Universal Robots PolyScope program: base_a.urp

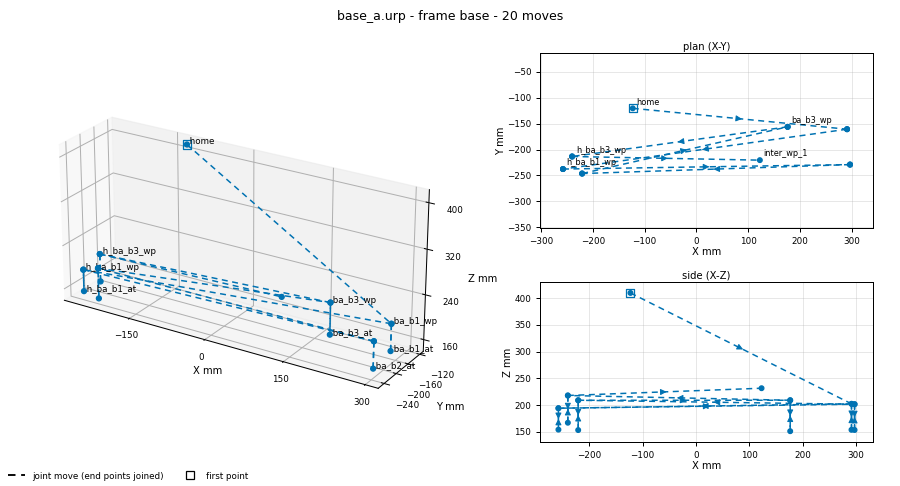
[picture p0: tool path of base_a.urp in frame base, 20 of 20 moves have a stored position in this frame; points joined in program order, loops and branches not executed]
Program base_a (installation=default directory=/programs/Session 1 createdIn=5.3.1.64192 lastSavedIn=5.3.1.64192 robotSerialNumber=20195300365)
Calibrated DH parameters: a=[-0.000093, -0.190649, -0.212673, 0.000091, -0.000205, 0]; d=[0.151591, 44.061648, -42.488068, -1.442789, 0.085322, 0.091911]; alpha=[1.570082, -0.003447, 0.007513, 1.572293, -1.571904, 0]; deltaTheta=[0, -0.672656, 0.728185, -0.055522, 0.000005, 0]
Robot Program (runOnlyOnce=true)
  URCap Gripper Activate (Robotiq_Grippers, Robotiq Inc.) dataModel(ResetAndActivateKey=false)
  URCap Gripper (Robotiq_Grippers, Robotiq Inc.) dataModel(position=50.0, force=100.0, speed=100.0, positionInDouble=50.0, forceInDouble=100.0, speedInDouble=100.0, slaveIds=[9], blocking=true)
  MoveJ speed 60 deg/s, acceleration 80 deg/s^2 (useActiveTCP=true) feature=Base
    Waypoint home: TCP in base x=-122.926 y=-120.377 z=410.038 mm, rx=2.273 ry=2.1657 rz=-0.0264 rad; joints [-85.876, -57.16, -80.452, -131.626, 89.649, -263.131] deg
  Folder Base_A
    MoveJ speed 60 deg/s, acceleration 80 deg/s^2 (useActiveTCP=true) feature=Base
      Waypoint ba_b1_wp: TCP in base x=291.339 y=-160.763 z=202.267 mm, rx=2.2196 ry=2.1634 rz=-0.046 rad; joints [-5.134, -97.09, -111.302, -60.85, 87.435, -183.275] deg
      Waypoint ba_b1_at: TCP in base x=291.327 y=-160.782 z=153.554 mm, rx=2.2196 ry=2.1633 rz=-0.046 rad; joints [-5.155, -104.362, -118.201, -46.683, 87.36, -183.222] deg
      URCap Gripper (Robotiq_Grippers, Robotiq Inc.) dataModel(position=100.0, force=100.0, speed=100.0, positionInDouble=100.0, forceInDouble=100.0, speedInDouble=100.0, slaveIds=[9], blocking=true)
      Waypoint ba_b1_wp: TCP in base x=291.339 y=-160.763 z=202.267 mm, rx=2.2196 ry=2.1634 rz=-0.046 rad; joints [-5.134, -97.09, -111.302, -60.85, 87.435, -183.275] deg
      Waypoint h_ba_b1_wp: TCP in base x=-257.858 y=-237.79 z=193.998 mm, rx=-3.1287 ry=0.0473 rz=-0.0059 rad; joints [-115.618, -102.966, -105.931, -61.783, 90.175, -203.494] deg
      Waypoint h_ba_b1_at: TCP in base x=-257.856 y=-237.787 z=153.878 mm, rx=-3.1287 ry=0.0473 rz=-0.006 rad; joints [-115.632, -108.549, -111.296, -50.837, 90.123, -203.451] deg
      URCap Gripper (Robotiq_Grippers, Robotiq Inc.) dataModel(position=50.0, force=100.0, speed=100.0, positionInDouble=50.0, forceInDouble=100.0, speedInDouble=100.0, slaveIds=[9], blocking=true)
      Waypoint h_ba_b1_wp: TCP in base x=-257.858 y=-237.79 z=193.998 mm, rx=-3.1287 ry=0.0473 rz=-0.0059 rad; joints [-115.618, -102.966, -105.931, -61.783, 90.175, -203.494] deg
    MoveJ speed 60 deg/s, acceleration 80 deg/s^2 (useActiveTCP=true) feature=Base
      Waypoint ba_b2_wp: TCP in base x=297.099 y=-229.137 z=201.509 mm, rx=2.2534 ry=2.1854 rz=-0.0426 rad; joints [-17.056, -107.569, -97.554, -65.462, 88.854, -194.942] deg
      Waypoint ba_b2_at: TCP in base x=297.093 y=-229.143 z=153.246 mm, rx=2.2534 ry=2.1854 rz=-0.0427 rad; joints [-17.073, -113.534, -103.963, -53.09, 88.799, -194.893] deg
      URCap Gripper (Robotiq_Grippers, Robotiq Inc.) dataModel(position=100.0, force=100.0, speed=100.0, positionInDouble=100.0, forceInDouble=100.0, speedInDouble=100.0, slaveIds=[9], blocking=true)
      Waypoint ba_b2_wp: TCP in base x=297.099 y=-229.137 z=201.509 mm, rx=2.2534 ry=2.1854 rz=-0.0426 rad; joints [-17.056, -107.569, -97.554, -65.462, 88.854, -194.942] deg
      Waypoint h_ba_b2_wp: TCP in base x=-220.82 y=-246.483 z=208.907 mm, rx=-3.1272 ry=0.0669 rz=0.002 rad; joints [-108.726, -96.552, -109.252, -64.858, 89.998, -195.885] deg
      Waypoint h_ba_b2_at: TCP in base x=-220.812 y=-246.497 z=153.058 mm, rx=-3.1273 ry=0.0669 rz=0.002 rad; joints [-108.744, -104.469, -117.433, -48.758, 89.918, -195.821] deg
      URCap Gripper (Robotiq_Grippers, Robotiq Inc.) dataModel(position=50.0, force=100.0, speed=100.0, positionInDouble=50.0, forceInDouble=100.0, speedInDouble=100.0, slaveIds=[9], blocking=true)
      Waypoint h_ba_b2_wp: TCP in base x=-220.82 y=-246.483 z=208.907 mm, rx=-3.1272 ry=0.0669 rz=0.002 rad; joints [-108.726, -96.552, -109.252, -64.858, 89.998, -195.885] deg
    MoveJ speed 60 deg/s, acceleration 80 deg/s^2 (useActiveTCP=true) feature=Base
      Waypoint ba_b3_wp: TCP in base x=176.479 y=-156.192 z=208.942 mm, rx=2.1987 ry=2.1726 rz=-0.0159 rad; joints [-7.147, -67.928, -134.317, -65.798, 88.131, -186.073] deg
      Waypoint ba_b3_at: TCP in base x=176.475 y=-156.198 z=150.955 mm, rx=2.1987 ry=2.1726 rz=-0.0159 rad; joints [-7.184, -79.69, -145.938, -42.419, 87.997, -185.98] deg
      URCap Gripper (Robotiq_Grippers, Robotiq Inc.) dataModel(position=100.0, force=100.0, speed=100.0, positionInDouble=100.0, forceInDouble=100.0, speedInDouble=100.0, slaveIds=[9], blocking=true)
      Waypoint ba_b3_wp: TCP in base x=176.479 y=-156.192 z=208.942 mm, rx=2.1987 ry=2.1726 rz=-0.0159 rad; joints [-7.147, -67.928, -134.317, -65.798, 88.131, -186.073] deg
      Waypoint h_ba_b3_wp: TCP in base x=-240.197 y=-213.51 z=217.855 mm, rx=2.242 ry=2.1952 rz=0.0362 rad; joints [-114.806, -93.519, -109.8, -67.774, 90.981, -293.227] deg
      Waypoint h_ba_b3_at: TCP in base x=-240.199 y=-213.502 z=166.817 mm, rx=2.242 ry=2.1953 rz=0.0361 rad; joints [-114.828, -100.186, -118.047, -52.858, 90.91, -293.168] deg
      URCap Gripper (Robotiq_Grippers, Robotiq Inc.) dataModel(position=50.0, force=100.0, speed=100.0, positionInDouble=50.0, forceInDouble=100.0, speedInDouble=100.0, slaveIds=[9], blocking=true)
      Waypoint h_ba_b3_wp: TCP in base x=-240.197 y=-213.51 z=217.855 mm, rx=2.242 ry=2.1952 rz=0.0362 rad; joints [-114.806, -93.519, -109.8, -67.774, 90.981, -293.227] deg
  MoveJ speed 60 deg/s, acceleration 80 deg/s^2 (useActiveTCP=true) feature=Base
    Waypoint inter_wp_1: TCP in base x=122.78 y=-220.583 z=231.495 mm, rx=2.2968 ry=2.1205 rz=-0.0201 rad; joints [-29.631, -72.124, -124.848, -72.343, 89.412, -204.687] deg
